{attribute 'qualified_only'}
{attribute 'strict'}
{attribute 'to_string'}
TYPE
ST128_TubeCapCheck_e :
(
    RESET := 0, // Reset

    INIT := 100, // Initialisieren 

    READY := 999,  // READY to Start, Init Done 
    START := 1000, // Start Zyklisch

    waitOnMover,     // wait until the mover is there
    MOVER_NEEDED_OP, // Ab here, a mover in position is needed to perform the action

    Move_shuttle_relative_right,
	Wait_move_and_check_tube_cap_right,
    Move_shuttle_to_pos_left,
	Wait_move_done_pos_left,
    Move_shuttle_relative_left,
	Wait_move_and_check_tube_cap_left,
    Save_result_in_mover,

    SYNC_MOVER_LEAVE, // MoverMan need to take the mover
    MOVER_FREE_OP,    // here, operation without mover can be done.

    DONE := 8000,  // Ablauf beendet 
    ERROR := 9000, // Fehler 
    _max
);
END_TYPE

(*
back to shuttle
check level NIO Box
*)

(* stored: Version 1.1.0.1, ProductVersion 3.1.4024.6
   EnumerationTextList ST128_TubeCapCheck_e: Id {0ef777c4-6dee-432f-a437-ff1bf8344346} *)
